TYPE ST_THROTTLE_VALVE :
STRUCT
	CURRENT_STATUS:DINT;
	CURRENT_CDG1_PRESSURE:DINT;(*1000Tor*)
	CURRENT_CDG2_PRESSURE:DINT;(*100Torr*)
	CURRENT_SET_PV:DINT;
	CURRENT_VALVE_POSITION:DINT;
	CURRENT_MODE:DINT;(*1: Pressure , 2:Position*)
	CURRENT_VALVE_MODE:DINT;
	
	SET_OUTPUT_MODE:DINT;
	SET_PRESSURE:DINT;
	SET_CONTROL_MODE:DINT;
	//1:Pressure Control, 2:Valve Position Control
END_STRUCT
END_TYPE

(* stored: Version 1.1.0.1, ProductVersion 3.1.4024.12
   DUT ST_THROTTLE_VALVE: Id {f8c856d0-9880-4a68-803a-88f0d5a9987b} *)
